PROGRAM P_Outputs_Manual
VAR
	//
	n_temp_speed_SP1: REAL;
	n_temp_speed_AP1: REAL;

END_VAR

//***********************************************************************************
//
// ETH Zürich / Robotic Fabrication Lab
// HIB C 13 / Stefano-Franscini-Platz 1
// CH-8093 Zürich
// 
// ***********************************************************************************
// 
// PROJECT     :  A061 Inline Mixer
// 
// FUNCTION    :  Outputs Manual Mode
// 
// AUTHOR      :  Fabio Scotto / Philippe Fleischmann / Weiting Chen
// 
// EMAIL       :  scotto@arch.ethz.ch / fleischmann@arch.ehtz.ch
// 
// Copyright   :  ETH Zürich (CH) 2022
//
// ***********************************************************************************


//***********************************************************************************
// Superplasticizer pump 1
//***********************************************************************************

//
// Power on
GVL_IO.ob_SP1_Power_On:=GVL_VAR.b_Mode_Manual;
//
// Pressure is Okay, always set it to True
GVL_IO.ob_SP1_Pressure_Ok:=TRUE;
//
// Bucket is not empty, always set it to true
GVL_IO.ob_SP1_Not_Empty:=TRUE;
//
// Pulse mode is a preset amount,  not in use
GVL_IO.ob_SP1_Pulse:=FALSE;


//
// Start pump
IF		P_SP1_OnOff.n_step= 30 
	OR 	P_SP1_Check.n_Step= 30 
THEN
	//
	// Pump On
	GVL_IO.ob_SP1_Start:=TRUE;
ELSE
	//
	// Pump On
	GVL_IO.ob_SP1_Start:=FALSE;
END_IF

//
// Speeds for Superplastizier pump
IF GVL_ResearchData.b_RED_Superplasticizer_Pump_Flush_On AND P_SP1_OnOff.n_step= 30 THEN
	//
	// Process speed for flushing or filling the pipe
	n_temp_speed_SP1:=GVL_ResearchData.n_RED_Superplasticizer_Pump_Flush_Flowrate;

ELSIF P_SP1_Check.n_Step=20 OR P_SP1_Check.n_Step=30 THEN 	
	//	
	// Check Flowrate for pump
	n_temp_speed_SP1:=GVL_ResearchData.n_RED_Superplasticizer_Pump_Check_Flowrate;
	
ELSE
	//
	// Process speed for pump
	n_temp_speed_SP1:=GVL_ResearchData.n_RED_Superplasticizer_Pump_Flowrate; // change to poti

END_IF

GVL_IO.on_SP1_Speed:=F_ScalAnalogOut(
	n_Input:= REAL_TO_INT(n_temp_speed_SP1),
	n_InMin:= 0, 
	n_InMax:= REAL_TO_INT(GVL_ResearchData.f_RED_Status_Superplasticizer_Pump_Max_Flowrate_ml_per_min), 
	n_OutMin:= 0, 
	n_OutMax:= 32767);


//***********************************************************************************
// Accelerator pump 1
//***********************************************************************************

//
// Power on
GVL_IO.ob_AP1_Power_On:=GVL_VAR.b_Mode_Manual;
//
// Pressure okey always set to true
GVL_IO.ob_AP1_Pressure_Ok:=TRUE;
//
// Bucket not empty always set to true
GVL_IO.ob_AP1_Not_Empty:=TRUE;
//
// Pulse a preset amount not in use
GVL_IO.ob_AP1_Pulse:=FALSE;

//
// Start pump
IF 	   P_AP1_OnOff.n_Step=30 
	OR P_AP1_Check.n_Step=30
THEN
	//
	// Pump on
	GVL_IO.ob_AP1_Start:=TRUE;
ELSE
	//
	// Pump off
	GVL_IO.ob_AP1_Start:=FALSE;
END_IF

//
// Speed for accelerator pump
IF GVL_ResearchData.b_RED_Acceleration_Pump_Flush_On AND P_AP1_OnOff.n_Step=30 THEN
	//
	// Process speed for flushing or filling the pipe
	n_temp_speed_AP1:=GVL_ResearchData.n_RED_Acceleration_Pump_Flush_Flowrate;
ELSIF P_AP1_Check.n_Step=20 OR P_AP1_Check.n_Step=30 THEN
	//	
	// Check Flowrate for pump
	n_temp_speed_AP1:=GVL_ResearchData.n_RED_Acceleration_Pump_Check_Flowrate;
ELSE
	//
	// Process speed for pump
	n_temp_speed_AP1:=GVL_IO.in_AP1_Poti_Speed;
END_IF

GVL_IO.on_AP1_Speed:=F_ScalAnalogOut(
	n_Input:= REAL_TO_INT(n_temp_speed_AP1),
	n_InMin:= 0, 
	n_InMax:= REAL_TO_INT(GVL_ResearchData.f_RED_Status_Acceleration_Pump_Max_Flowrate_ml_per_min), 
	n_OutMin:= 0, 
	n_OutMax:= 32767);


// ***********************************************************************************
// Concrete Pump 1 
// ***********************************************************************************

//
// Start
IF  P_CP1_Enable.n_Step=20 THEN
	GVL_IO.ob_CP1_Start:=TRUE;
ELSE
	GVL_IO.ob_CP1_Start:=FALSE;
END_IF

//
// Stop
IF  P_CP1_Enable.n_Step=40 THEN
	GVL_IO.ob_CP1_Stop:=TRUE;
ELSE
	GVL_IO.ob_CP1_Stop:=FALSE;
END_IF

//
// Forward
GVL_IO.ob_CP1_Forward:=GVL_ResearchData.b_RED_Concrete_Pump_Forward_On;

//
// Backward
GVL_IO.ob_CP1_Backward:=GVL_ResearchData.b_RED_Concrete_Pump_Backward_On;

//
// Concrete pump speed  0 (0V) to 75 rpm (10V)
GVL_IO.on_CP1_Speed:=F_ScalAnalogOut(
	n_Input:=GVL_ResearchData.n_RED_Concrete_Pump_Speed, 
	n_InMin:=0, 
	n_InMax:=75, 
	n_OutMin:=0, 
	n_OutMax:=32767);

END_PROGRAM

(* stored: Version 1.1.0.1, ProductVersion 3.1.4024.11
   POU P_Outputs_Manual: Id {29a9fa82-67db-4e62-a260-6977b4aa95ba}, SpecialFunc None *)
